TYPE GestioneEncoderEsterno :
STRUCT
	Azzera : BOOL; //Comando di azzeramento encoder
	Pronto : BOOL; //Stato di encoder Pronto
	Direzione : bool; //Direzione di conteggio
END_STRUCT
END_TYPE

(* stored: Version 1.1.0.1, ProductVersion 3.1.4024.11
   DUT GestioneEncoderEsterno: Id {3bbfcc20-1780-4359-9e5e-4af3b949d099} *)
